FUNCTION_BLOCK DIO_IN_4CH (* Service Interface Function Block Type *)
  (* Standard: 61499-2 *)
  (* Version 0.0, 07/06/2021, josef, nxtControl GmBH, template *)
  PACKAGE Flexbridge.Iceblock;
  (* Compiler Cpp nxtControl builtin 1.0 *)
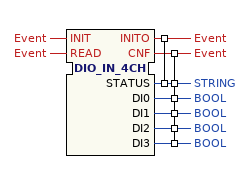
  EVENT_INPUT
    INIT;
    READ;
  END_EVENT
  EVENT_OUTPUT
    INITO WITH STATUS;
    CNF WITH STATUS, DI0, DI1, DI2, DI3;
  END_EVENT
  VAR_OUTPUT
    STATUS : STRING;
    DI0 : BOOL;
    DI1 : BOOL;
    DI2 : BOOL;
    DI3 : BOOL;
  END_VAR
  SERVICE DIO_IN/RESOURCE
    SEQUENCE normal_establishment
      DIO_IN.INIT+(PARAMS) -> RESOURCE.initialize(PARAMS) -> DIO_IN.INITO+();
    END_SEQUENCE
    SEQUENCE unsuccessful_establishment
      DIO_IN.INIT+(PARAMS) -> RESOURCE.initialize(PARAMS) -> DIO_IN.INITO-(STATUS);
    END_SEQUENCE
    SEQUENCE request_confirm
      DIO_IN.REQ+(SD) -> RESOURCE.request(SD) -> DIO_IN.CNF+(RD);
    END_SEQUENCE
    SEQUENCE request_inhibited
      DIO_IN.REQ-(SD) -> DIO_IN.CNF-(STATUS);
    END_SEQUENCE
    SEQUENCE request_error
      DIO_IN.REQ+(SD) -> RESOURCE.request(SD) -> DIO_IN.CNF-(STATUS);
    END_SEQUENCE
    SEQUENCE indication_response
      RESOURCE.indicate(RD) -> DIO_IN.IND+(RD);
      DIO_IN.RSP(QI,SD) -> RESOURCE.response(QI,SD);
    END_SEQUENCE
    SEQUENCE indication_inhibited
      RESOURCE.indicate(RD,QI=FALSE) -> RESOURCE.inhibited();
    END_SEQUENCE
    SEQUENCE error_indication
      RESOURCE.error(STATUS) -> DIO_IN.IND-(STATUS);
    END_SEQUENCE
    SEQUENCE application_initiated_termination
      DIO_IN.INIT-() -> RESOURCE.terminate() -> DIO_IN.INITO-(STATUS);
    END_SEQUENCE
    SEQUENCE resource_initiated_termination
      -> DIO_IN.INITO-(STATUS);
    END_SEQUENCE
  END_SERVICE
END_FUNCTION_BLOCK
